{attribute 'GeneratedUsingTerminal: EK1100-0000-0018'}
{attribute addProperty BoxType "EK1100-0000-0018"}
{attribute addProperty Id "TcTerminals210_2BK1250TcTerminals210_2BK1250_CEF741550"}
{attribute addProperty CRC "1354842929"}
{attribute addProperty Size "0"}
TYPE TcTerminals210_2EK1100_50C14331 EXTENDS EK1100_1FC0878B :
STRUCT
	{attribute addProperty Name "TcTerminals210_2BK1250"}
	{attribute addProperty PreviousPort "TcTerminals210_2EK1100 : B"}
	TcTerminals210_2BK1250 : TcTerminals210_2BK1250_CEF74155;
END_STRUCT
END_TYPE

(* stored: Version 1.2.0.0, ProductVersion 3.1.4024.9
   DUT TcTerminals210_2EK1100_50C14331: Id {57e22e18-4f30-47ee-992f-e121ae961f1b} *)
